{attribute 'qualified_only'}
{attribute 'strict'}
TYPE eCoolingPowerRequest :
(
	off := 0,
	intern := 1,
	full := 2
);
END_TYPE

(* stored: Version 1.1.0.1, ProductVersion 3.1.4024.12
   DUT eCoolingPowerRequest: Id {f6809b30-140c-4752-ad6f-d6928ca0db69} *)
